//{attribute 'qualified_only'}
VAR_GLOBAL
	
	pFEEDER_BULLET_PUSHER:  FB_PISTON;
	pFEEDER_HOLD1: FB_PISTON;
	pFEEDER_HOLD2: FB_PISTON;
	pFEEDER_OPEN1: FB_PISTON;
	pFEEDER_OPEN2: FB_PISTON;
	
	pSEPARATE1_LIFT:   FB_PISTON;
	pSEPARATE1_COLET1: FB_PISTON;
	pSEPARATE1_COLET2: FB_PISTON;
	pSEPARATE1_COLET3: FB_PISTON;
	pSEPARATE1_COLET4: FB_PISTON;
	pSEPARATE1_PUSHER_FROM_COLET1:  FB_PISTON;
	pSEPARATE1_PUSHER_FROM_COLET2:  FB_PISTON;
	pSEPARATE1_DRAWER:  FB_PISTON;
	pSEPARATE1_DRAWER_PUSHER:  FB_PISTON;
	pSEPARATE1_DRAWER_DOOR:  FB_PISTON;
	
	pSEPARATE2_LIFT:   FB_PISTON;
	pSEPARATE2_COLET1: FB_PISTON;
	pSEPARATE2_COLET2: FB_PISTON;
	pSEPARATE2_COLET3: FB_PISTON;
	pSEPARATE2_COLET4: FB_PISTON;
	pSEPARATE2_PUSHER_FROM_COLET1:  FB_PISTON;
	pSEPARATE2_PUSHER_FROM_COLET2:  FB_PISTON;
	pSEPARATE2_DRAWER:  FB_PISTON;
	pSEPARATE2_DRAWER_PUSHER:  FB_PISTON;
	pSEPARATE2_DRAWER_DOOR:  FB_PISTON;
	
	pVERIFICATION_OPEN1: FB_PISTON;
	pVERIFICATION_OPEN2: FB_PISTON;
	
	pCLEANER_PISTON: FB_PISTON;
	pCLEANER_AIR: FB_PISTON;
	
	pPRIMER_1: FB_PISTON;
	pPRIMER_2: FB_PISTON;
	
	pRELEASE_OPEN1: FB_PISTON;
	pRELEASE_OPEN2: FB_PISTON;
	pRELEASE_PUSHER: FB_PISTON;
	
	
	
	
	
END_VAR

(* stored: Version 1.1.0.1, ProductVersion 3.1.4024.12
   GVL GVL_PISTONS: Id {bf755774-5f2d-4774-a60c-afb3556ed773} *)
